FUNCTION_BLOCK Test_F_TimeAsString_ReturnsLeadingZeros EXTENDS T_UnitTestBase
VAR
    TimeStruct : TIMESTRUCT := (wHour := 6, wMinute := 5, wSecond := 4);
END_VAR

METHOD Init
VAR_INPUT
END_VAR
END_METHOD

{attribute 'analysis' := '-33'} // inhibit unused variable warning
METHOD RunTest
AssertEquals_STRING(Expected := '06:05:04',
                    Actual   := F_TimeAsString(TimeStruct),
                    Message  := 'F_TimeAsString(TimeStruct)');

TestCompleted := TRUE;
END_METHOD

END_FUNCTION_BLOCK

(* stored: Version 1.1.0.1, ProductVersion 3.1.4024.12
   POU Test_F_TimeAsString_ReturnsLeadingZeros: Id {72a01420-e5e9-02f9-2a71-637672ec7977}, SpecialFunc None
   Method Init: Id {40260e9e-96b8-084c-39b3-010d9d525b1d}
   Method RunTest: Id {6dcac63e-26da-04c2-3387-6790f1d49358} *)
